# EPICS autosave request: quadEMApp/Db/NSLS2_EM_settings.req
$(P)$(R)ADCOffset1
$(P)$(R)ADCOffset2
$(P)$(R)ADCOffset3
$(P)$(R)ADCOffset4
